// TIA Portal V17 export
// export: Created 2023-04-11T09:34:00.7441836Z, ExportSetting WithDefaults, DisplayName Totally Integrated Automation Portal, DisplayVersion V17 Update 3, DisplayName TIA Portal Openness, DisplayVersion V17 Update 3, DisplayName TIA Portal Version Control Interface, DisplayVersion V17, DisplayName SINAMICS Startdrive Advanced, DisplayVersion V17 Update2, DisplayName SINAMICS Startdrive G130, G150, S120, S150, SINAMICS MV, S210, DisplayVersion V17 Update2, DisplayName SINAMICS Startdrive G110M, G120, G120C, G120D, G120P, G115D, DisplayVersion V17 Update2, DisplayName STEP 7 Professional, DisplayVersion V17 Update 3, DisplayName STEP 7 Safety, DisplayVersion V17, DisplayName WinCC UA Professional, DisplayVersion V17 Update 3
FUNCTION "FC_int2str_1" : Void   // FC48, LAD
{ S7_Optimized_Access := 'TRUE' }
VERSION : 0.1
// stored: AutoNumber true, IsIECCheckEnabled false, SetENOAutomatically false, UDAEnableTagReadback false
   VAR_INPUT
      In : Int;
   END_VAR
   VAR_OUTPUT
      Out : String;
   END_VAR
   VAR_TEMP
      auxStr : String;
   END_VAR
   VAR_TEMP   // added for the SCL form of the ladder/FBD networks
      _w1 : Bool;
   END_VAR
BEGIN

REGION Network 1: Init conversion string
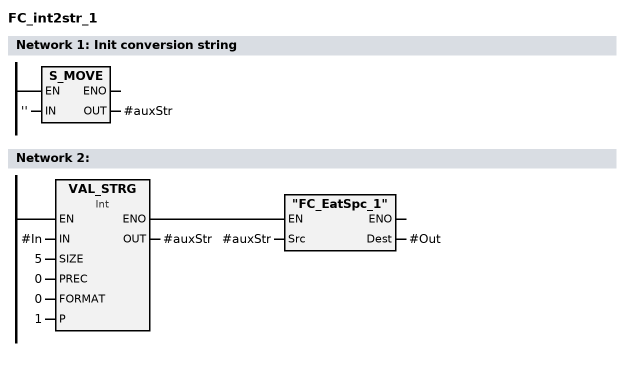
   RUNG wire#powerrail
      S_Move(in := '', out => #auxStr)
   END_RUNG
   // the same network as SCL:
   #auxStr := '';
END_REGION

REGION Network 2
   RUNG wire#powerrail
      { S7_Templates := "[value_type := Int, str_type := String]" } VAL_STRG(IN := #In, SIZE := 5, PREC := 0, FORMAT := 0, P := 1, OUT => #auxStr)
      "FC_EatSpc_1"(Src := #auxStr, Dest => #Out)
   END_RUNG
   // the same network as SCL:
   VAL_STRG(IN := #In, SIZE := 5, PREC := 0, FORMAT := 0, P := 1, OUT => #auxStr, ENO => #_w1);
   IF #_w1 THEN "FC_EatSpc_1"(Src := #auxStr, Dest => #Out); END_IF;
END_REGION
END_FUNCTION
